// Mitsubishi GX Works2 project: GX W2 L2 Ex 5 DK c   PLC: FX3G

// global labels: Global1
VAR_GLOBAL
  iFan AT Y001 : BOOL;
END_VAR

// task Task_01 (event TRUE, interval 0, priority 31): POU_01

PROGRAM POU_01
VAR
  Pulse_Timer1 : TP;
  bStart : BOOL;
END_VAR
(* structured ladder/FBD written out as ST: instructions are called as NAME(EN, inputs, outputs); _pN, _eN, _tN stand for wires *)
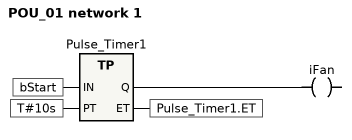
(* network 1 *)
Pulse_Timer1(IN := bStart, PT := T#10s, ET => Pulse_Timer1.ET);
iFan := Pulse_Timer1.Q;
END_PROGRAM
